// TIA Portal V16 export
// export: Created 2021-03-04T22:03:59.3995966Z, ExportSetting WithDefaults, DisplayName Totally Integrated Automation Portal, DisplayVersion V16, DisplayName TIA Portal Version Control Interface, DisplayVersion V16, DisplayName TIA Portal Openness, DisplayVersion V16, DisplayName SINAMICS Startdrive Advanced, DisplayVersion V16, DisplayName SINAMICS Startdrive G130, G150, S120, S150, SINAMICS MV, S210, DisplayVersion V16, DisplayName SINAMICS Startdrive G110M, G120, G120C, G120D, G120P, DisplayVersion V16, DisplayName STEP 7 Professional, DisplayVersion V16, DisplayName STEP 7 Safety, DisplayVersion V16, DisplayName WinCC Professional, DisplayVersion V16
FUNCTION_BLOCK "fbRack"   // FB5, LAD
{ S7_Optimized_Access := 'TRUE' }
VERSION : 0.1
// stored: AutoNumber true, IsIECCheckEnabled false, IsRetainMemResEnabled false, MemoryReserve 100, SetENOAutomatically false, UDAEnableTagReadback false
   VAR_INPUT
      iInMutexLockConfirmation { ExternalAccessible := 'False'; ExternalVisible := 'False'; ExternalWritable := 'False'} : Int;
      udtInLastNutrientReading { ExternalAccessible := 'False'; ExternalVisible := 'False'; ExternalWritable := 'False'} : "udtNutrientReading";
      bInSupplySolenoidFromRoomFertigation { ExternalAccessible := 'False'; ExternalVisible := 'False'; ExternalWritable := 'False'} : Bool;
      bInReturnSolenoidFromRoomFertigation { ExternalAccessible := 'False'; ExternalVisible := 'False'; ExternalWritable := 'False'} : Bool;
      iInLightsDelaySecs { ExternalAccessible := 'False'; ExternalVisible := 'False'; ExternalWritable := 'False'} : Int;
      rInCurrentTemperature : Real;
      arrAI { ExternalAccessible := 'False'; ExternalVisible := 'False'; ExternalWritable := 'False'} : Array[1.."NUM_AI_RACK"] of Int;
      AI AT arrAI : "udtRackAI";
   END_VAR
   VAR_OUTPUT
      iOutMutexRequest { ExternalAccessible := 'False'; ExternalVisible := 'False'; ExternalWritable := 'False'} : Int;
      OutFertigationSettings { ExternalAccessible := 'False'; ExternalVisible := 'False'; ExternalWritable := 'False'} : "udtFertigationSettings";
      arrDQ { ExternalAccessible := 'False'; ExternalVisible := 'False'; ExternalWritable := 'False'} : Array[1.."NUM_DQ_RACK"] of Bool;
      DQ AT arrDQ : "udtRackDQ";
   END_VAR
   VAR
      Lighting { ExternalVisible := 'False'} : "fbRackLights";
      Fertigation { ExternalVisible := 'False'} : "fbRackFertigation";
      AI_ReservoirLevel { ExternalVisible := 'False'} : "fbAlarmedSetpoint";
   END_VAR
   VAR RETAIN
      DQ_SupplySolenoid { ExternalVisible := 'False'} : "udtDigitalOutput";
      DQ_ReturnSolenoid { ExternalVisible := 'False'} : "udtDigitalOutput";
      DQ_ShelfSolenoid { ExternalVisible := 'False'} : "udtDigitalOutput";
      DQ_Lights { ExternalVisible := 'False'} : "udtDigitalOutput";
   END_VAR
   // AI_ReservoirLevel.Config.rLowCalibration := 0.0;
   // AI_ReservoirLevel.Config.rHighCalibration := 951.0;
BEGIN

REGION Network 1 (SCL)
   // Note that rack supply/return solenoids are managed by room-level fertigation FB
   // Process rack-level analog inputs
   #AI_ReservoirLevel(#AI.IW_ReservoirLevel);

   // Call lighting control fb
   #Lighting(iInDelaySecs := #iInLightsDelaySecs,
             rInCurrentTemperature := #rInCurrentTemperature,
             bOutLights => #Lighting.bOutLights);

   // Call rack-level fertigation logic
   #Fertigation(iInMutexLockConfirmation := #iInMutexLockConfirmation,
                InLastNutrientReading:= #udtInLastNutrientReading,
                rInReservoirLevel := #AI_ReservoirLevel.rActual,
                bInReturnSolenoidStatus:=#DQ.Q_ReturnSolenoid,
                bInShelfSolenoidStatus:=#DQ.Q_ShelfSolenoid,
                iOutMutexRequest => #iOutMutexRequest,
                OutFertigationSettings => #OutFertigationSettings,
                bOutShelfSolenoid => #Fertigation.bOutShelfSolenoid);

   // Set rack-level outputs
   // Rack supply/return solenoids are managed by room-level fertigation FB
   #DQ.Q_SupplySolenoid := "fcDigitalOutput"(bInAutoVal := #bInSupplySolenoidFromRoomFertigation, InOutUdt := #DQ_SupplySolenoid);
   #DQ.Q_ReturnSolenoid := "fcDigitalOutput"(bInAutoVal := #bInReturnSolenoidFromRoomFertigation, InOutUdt := #DQ_ReturnSolenoid);
   #DQ.Q_ShelfSolenoid  := "fcDigitalOutput"(bInAutoVal := #Fertigation.bOutShelfSolenoid, InOutUdt := #DQ_ShelfSolenoid);
   #DQ.Q_Lights         := "fcDigitalOutput"(bInAutoVal := #Lighting.bOutLights, InOutUdt := #DQ_Lights);
END_REGION
END_FUNCTION_BLOCK
